Omron CX-Programmer project NewProject (CX-Programmer 9.75)

# PLC NewPLC1: CP2E-N N

## Global symbols (name address type ; comment)
modbus _CP2E003_ExecuteModTcpServer

## Program NewProgram1 (cyclic task 0)
Local symbols
P_ON BOOL
p_on BOOL

### Section Section1

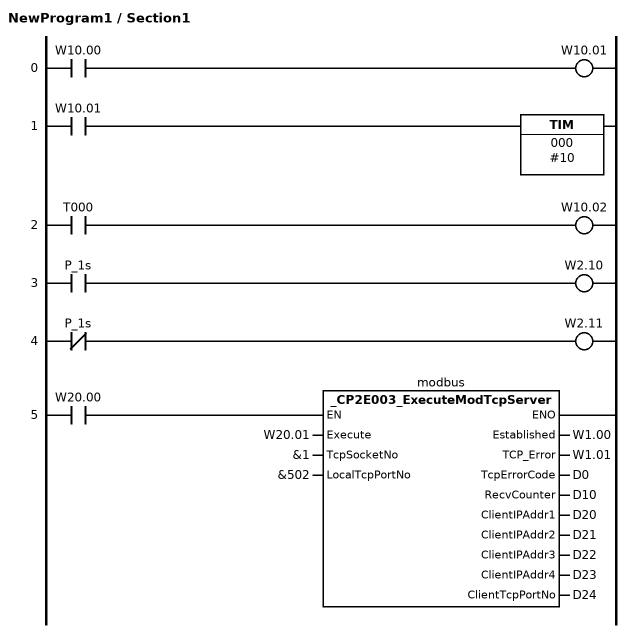
; rung 0
LD W10.00
OUT W10.01
; rung 1
LD W10.01
TIM 000 #10
; rung 2
LD T000
OUT W10.02
; rung 3
LD P_1s
OUT W2.10
; rung 4
LDNOT P_1s
OUT W2.11
; rung 5
LD W20.00
CALL modbus : _CP2E003_ExecuteModTcpServer (Execute := W20.01, TcpSocketNo := &1, LocalTcpPortNo := &502, Established => W1.00, TCP_Error => W1.01, TcpErrorCode => D0, RecvCounter => D10, ClientIPAddr1 => D20, ClientIPAddr2 => D21, ClientIPAddr3 => D22, ClientIPAddr4 => D23, ClientTcpPortNo => D24)

### Section END
; rung 0
END(001)

## Function block _CP2E003_ExecuteModTcpServer (Omron library block, body left out)